{attribute 'GeneratedUsingTerminal: EP2316-0008-0017'}
{attribute addProperty BoxType "EP2316-0008-0017"}
{attribute addProperty Id "InputAT %I*ARRAY[0..7] OF BOOL8Sync_ErrorAT %I*BOOL1"}
{attribute addProperty CRC "2788215981"}
{attribute addProperty Size "9"}
TYPE DO_Diag_Inputs_CC455148 EXTENDS InputBase_8311D824 :
STRUCT
	{attribute addProperty Name "Input"}
	Input AT %I* : ARRAY[0..7] OF BOOL;
	{attribute addProperty Name "Sync_Error"}
	Sync_Error AT %I* : BOOL;
END_STRUCT
END_TYPE

(* stored: Version 1.2.0.0, ProductVersion 3.1.4024.11
   DUT DO_Diag_Inputs_CC455148: Id {05e3e1a5-9411-4860-aab0-beee64b64814} *)
